(* IEC 61131-3 sources: Lasal/CPU_5344_V01/Class/OperationDataV2, 1 file *)

(* ---- OperationDataV2.st ---- *)
(*!
<Class
	Name               = "OperationDataV2"
	Revision           = "0.0"
	RealtimeTask       = "false"
	CyclicTask         = "false"
	BackgroundTask     = "false"
	Sigmatek           = "false"
	OSInterface        = "false"
	HighPriority       = "false"
	Automatic          = "false"
	UpdateMode         = "Prescan"
	SharedCommandTable = "true"
	Objectsize         = "(450,120)">
	<Channels>
		<Server Name="ClassSvr" Visualized="false" Initialize="false" WriteProtected="true" Retentive="false"/>
		<Server Name="firstIdx" Visualized="true" Initialize="false" WriteProtected="false" Retentive="false"/>
		<Client Name="BewLine1" Required="true" Internal="true"/>
		<Client Name="BewLine2" Required="true" Internal="true"/>
		<Client Name="BewLine3" Required="true" Internal="true"/>
		<Client Name="BewLine4" Required="true" Internal="true"/>
		<Client Name="BewLine5" Required="true" Internal="true"/>
		<Client Name="BewLine6" Required="true" Internal="true"/>
		<Client Name="Line1" Required="true" Internal="true"/>
		<Client Name="Line2" Required="true" Internal="true"/>
		<Client Name="Line3" Required="true" Internal="true"/>
		<Client Name="Line4" Required="true" Internal="true"/>
		<Client Name="Line5" Required="true" Internal="true"/>
		<Client Name="Line6" Required="true" Internal="true"/>
	</Channels>
	<Network Name="OperationDataV2">
		<!-- List of Components in this network -->
		<Components>
			<Object
				Name       = "BewLine1"
				Class      = "tMyBDintTODint"
				Position   = "(150,870)"
				Visualized = "true">
				<Channels>
					<Server Name="ClassSvr"/>
					<Server Name="Data"/>
					<Client Name="cOutput"/>
				</Channels>
			</Object>
			<Object
				Name       = "BewLine2"
				Class      = "tMyBDintTODint"
				Position   = "(690,870)"
				Visualized = "true">
				<Channels>
					<Server Name="ClassSvr"/>
					<Server Name="Data"/>
					<Client Name="cOutput"/>
				</Channels>
			</Object>
			<Object
				Name       = "BewLine3"
				Class      = "tMyBDintTODint"
				Position   = "(1230,870)"
				Visualized = "true">
				<Channels>
					<Server Name="ClassSvr"/>
					<Server Name="Data"/>
					<Client Name="cOutput"/>
				</Channels>
			</Object>
			<Object
				Name       = "BewLine4"
				Class      = "tMyBDintTODint"
				Position   = "(1770,870)"
				Visualized = "true">
				<Channels>
					<Server Name="ClassSvr"/>
					<Server Name="Data"/>
					<Client Name="cOutput"/>
				</Channels>
			</Object>
			<Object
				Name       = "BewLine5"
				Class      = "tMyBDintTODint"
				Position   = "(2340,870)"
				Visualized = "true">
				<Channels>
					<Server Name="ClassSvr"/>
					<Server Name="Data"/>
					<Client Name="cOutput"/>
				</Channels>
			</Object>
			<Object
				Name       = "BewLine6"
				Class      = "tMyBDintTODint"
				Position   = "(2910,870)"
				Visualized = "true">
				<Channels>
					<Server Name="ClassSvr"/>
					<Server Name="Data"/>
					<Client Name="cOutput"/>
				</Channels>
			</Object>
			<Object
				Name       = "Line1"
				Class      = "OperationLineV2"
				Position   = "(150,270)"
				Visualized = "true">
				<Channels>
					<Server Name="amount"/>
					<Server Name="ClassSvr"/>
					<Server Name="operationId"/>
					<Server Name="operationType"/>
					<Server Name="pitch"/>
					<Server Name="rnr"/>
					<Server Name="xPos"/>
					<Server Name="yPos"/>
					<Server Name="zPos"/>
				</Channels>
			</Object>
			<Object
				Name       = "Line2"
				Class      = "OperationLineV2"
				Position   = "(690,270)"
				Visualized = "true">
				<Channels>
					<Server Name="amount"/>
					<Server Name="ClassSvr"/>
					<Server Name="operationId"/>
					<Server Name="operationType"/>
					<Server Name="pitch"/>
					<Server Name="rnr"/>
					<Server Name="xPos"/>
					<Server Name="yPos"/>
					<Server Name="zPos"/>
				</Channels>
			</Object>
			<Object
				Name       = "Line3"
				Class      = "OperationLineV2"
				Position   = "(1230,270)"
				Visualized = "true">
				<Channels>
					<Server Name="amount"/>
					<Server Name="ClassSvr"/>
					<Server Name="operationId"/>
					<Server Name="operationType"/>
					<Server Name="pitch"/>
					<Server Name="rnr"/>
					<Server Name="xPos"/>
					<Server Name="yPos"/>
					<Server Name="zPos"/>
				</Channels>
			</Object>
			<Object
				Name       = "Line4"
				Class      = "OperationLineV2"
				Position   = "(1770,270)"
				Visualized = "true">
				<Channels>
					<Server Name="amount"/>
					<Server Name="ClassSvr"/>
					<Server Name="operationId"/>
					<Server Name="operationType"/>
					<Server Name="pitch"/>
					<Server Name="rnr"/>
					<Server Name="xPos"/>
					<Server Name="yPos"/>
					<Server Name="zPos"/>
				</Channels>
			</Object>
			<Object
				Name       = "Line5"
				Class      = "OperationLineV2"
				Position   = "(2340,270)"
				Visualized = "true">
				<Channels>
					<Server Name="amount"/>
					<Server Name="ClassSvr"/>
					<Server Name="operationId"/>
					<Server Name="operationType"/>
					<Server Name="pitch"/>
					<Server Name="rnr"/>
					<Server Name="xPos"/>
					<Server Name="yPos"/>
					<Server Name="zPos"/>
				</Channels>
			</Object>
			<Object
				Name       = "Line6"
				Class      = "OperationLineV2"
				Position   = "(2910,270)"
				Visualized = "true">
				<Channels>
					<Server Name="amount"/>
					<Server Name="ClassSvr"/>
					<Server Name="operationId"/>
					<Server Name="operationType"/>
					<Server Name="pitch"/>
					<Server Name="rnr"/>
					<Server Name="xPos"/>
					<Server Name="yPos"/>
					<Server Name="zPos"/>
				</Channels>
			</Object>
		</Components>
		<Comments>
		</Comments>
		<!-- List of Connections in this network -->
		<Connections>
			<Connection Source="this.Line1" Destination="Line1.ClassSvr"/>
			<Connection Source="this.Line2" Destination="Line2.ClassSvr"/>
			<Connection Source="this.Line3" Destination="Line3.ClassSvr"/>
			<Connection Source="this.Line4" Destination="Line4.ClassSvr"/>
			<Connection Source="this.Line5" Destination="Line5.ClassSvr"/>
			<Connection Source="this.Line6" Destination="Line6.ClassSvr"/>
			<Connection Source="this.BewLine1" Destination="BewLine1.ClassSvr"/>
			<Connection Source="BewLine1.cOutput" Destination="Line1.operationType" Vertices="(150,960),(556,780),"/>
			<Connection Source="this.BewLine2" Destination="BewLine2.ClassSvr"/>
			<Connection Source="this.BewLine5" Destination="BewLine5.ClassSvr"/>
			<Connection Source="this.BewLine3" Destination="BewLine3.ClassSvr"/>
			<Connection Source="BewLine6.cOutput" Destination="Line6.operationType" Vertices="(2910,960),(3316,780),"/>
			<Connection Source="this.BewLine4" Destination="BewLine4.ClassSvr"/>
			<Connection Source="BewLine5.cOutput" Destination="Line5.operationType" Vertices="(2340,960),(2746,780),"/>
			<Connection Source="this.BewLine6" Destination="BewLine6.ClassSvr"/>
			<Connection Source="BewLine4.cOutput" Destination="Line4.operationType" Vertices="(1770,960),(2176,780),"/>
			<Connection Source="BewLine3.cOutput" Destination="Line3.operationType" Vertices="(1230,960),(1636,780),"/>
			<Connection Source="BewLine2.cOutput" Destination="Line2.operationType" Vertices="(690,960),(1096,780),"/>
		</Connections>
		<!-- Headerfiles -->
		<Options>
		</Options>
	</Network>
</Class>
*)
OperationDataV2 : CLASS
  //Servers:
	ClassSvr 	: SvrChCmd_DINT;
	firstIdx 	: SvrCh_DINT;
  //Clients:
	BewLine1 	: CltChCmd_tMyBDintTODint;
	BewLine2 	: CltChCmd_tMyBDintTODint;
	BewLine3 	: CltChCmd_tMyBDintTODint;
	BewLine4 	: CltChCmd_tMyBDintTODint;
	BewLine5 	: CltChCmd_tMyBDintTODint;
	BewLine6 	: CltChCmd_tMyBDintTODint;
	Line1 	: CltChCmd_OperationLineV2;
	Line5 	: CltChCmd_OperationLineV2;
	Line4 	: CltChCmd_OperationLineV2;
	Line3 	: CltChCmd_OperationLineV2;
	Line2 	: CltChCmd_OperationLineV2;
	Line6 	: CltChCmd_OperationLineV2;
  //Variables:
		actPtr 	: ^ProductsDbV2::tRecipeLineList;
		actPtrHeigth 	: ^DINT;
		actUseHeigth 	: DINT;
		dbMaxLines 	: DINT;
  //Functions:

	FUNCTION GLOBAL WritePtrs
		VAR_INPUT
			ptr 	: ^ProductsDbV2::tRecipeLineList;
			ptrProdHeigth 	: ^DINT;
			useHeigth 	: DINT;
			maxLines 	: DINT;
		END_VAR;

	FUNCTION VIRTUAL GLOBAL firstIdx::Write
		VAR_INPUT
			input (EAX) 	: DINT;
		END_VAR
		VAR_OUTPUT
			result (EAX) 	: DINT;
		END_VAR;
  //Tables:
	FUNCTION @STD
		VAR_OUTPUT
			ret_code	: CONFSTATES;
		END_VAR;
	FUNCTION GLOBAL TAB @CT_;
END_CLASS;

#pragma using OperationLineV2
#pragma using tMyBDintTODint

FUNCTION GLOBAL OperationDataV2::WritePtrs
	VAR_INPUT
		ptr 	: ^ProductsDbV2::tRecipeLineList;
		ptrProdHeigth 	: ^DINT;
		useHeigth 	: DINT;
		maxLines 	: DINT;
	END_VAR

  actPtr := ptr;
  actPtrHeigth := ptrProdHeigth;
  actUseHeigth := useHeigth;
  dbMaxLines := maxLines;

  Line1.WritePtr(iptr:=#actPtr^[0], iPtrProdHeigth:=ptrProdHeigth, iUseHeigth:=useHeigth);
  Line2.WritePtr(iptr:=#actPtr^[1], iPtrProdHeigth:=ptrProdHeigth, iUseHeigth:=useHeigth);
  Line3.WritePtr(iptr:=#actPtr^[2], iPtrProdHeigth:=ptrProdHeigth, iUseHeigth:=useHeigth);
  Line4.WritePtr(iptr:=#actPtr^[3], iPtrProdHeigth:=ptrProdHeigth, iUseHeigth:=useHeigth);
  Line5.WritePtr(iptr:=#actPtr^[4], iPtrProdHeigth:=ptrProdHeigth, iUseHeigth:=useHeigth);
  Line6.WritePtr(iptr:=#actPtr^[5], iPtrProdHeigth:=ptrProdHeigth, iUseHeigth:=useHeigth);
  Line1.rnr:= 1;
  Line2.rnr:= 2;
  Line3.rnr:= 3;
  Line4.rnr:= 4;
  Line5.rnr:= 5;
  Line6.rnr:= 6;

END_FUNCTION

FUNCTION VIRTUAL GLOBAL OperationDataV2::firstIdx::Write
	VAR_INPUT
		input (EAX) 	: DINT;
	END_VAR
	VAR_OUTPUT
		result (EAX) 	: DINT;
	END_VAR

	firstIdx := input;

  if firstIdx >= 0 & firstIdx < (dbMaxLines-5) & actPtr<>NIL then
    Line1.WritePtr(iptr:=#actPtr^[firstIdx], iPtrProdHeigth:=actPtrHeigth, iUseHeigth:=actUseHeigth);
    Line1.rnr := firstIdx + 1;

    Line2.WritePtr(iptr:=#actPtr^[firstIdx+1], iPtrProdHeigth:=actPtrHeigth, iUseHeigth:=actUseHeigth);
    Line2.rnr := firstIdx + 2;

    Line3.WritePtr(iptr:=#actPtr^[firstIdx+2], iPtrProdHeigth:=actPtrHeigth, iUseHeigth:=actUseHeigth);
    Line3.rnr := firstIdx +3;

    Line4.WritePtr(iptr:=#actPtr^[firstIdx+3], iPtrProdHeigth:=actPtrHeigth, iUseHeigth:=actUseHeigth);
    Line4.rnr := firstIdx +4;

    Line5.WritePtr(iptr:=#actPtr^[firstIdx+4], iPtrProdHeigth:=actPtrHeigth, iUseHeigth:=actUseHeigth);
    Line5.rnr := firstIdx +5;

    Line6.WritePtr(iptr:=#actPtr^[firstIdx+5], iPtrProdHeigth:=actPtrHeigth, iUseHeigth:=actUseHeigth);
    Line6.rnr := firstIdx +6;

  else
    result := ACCESS_DENIED;
  end_if;

	result := firstIdx;

END_FUNCTION
